TYPE ST_EL3174 :
STRUCT
	Ch1_Error						AT %I*	:BOOL;
	Ch1_Value						AT %I*	:INT;
	Ch2_Error						AT %I*	:BOOL;
	Ch2_Value						AT %I*	:INT;
	Ch3_Error						AT %I*	:BOOL;
	Ch3_Value						AT %I*	:INT;
	Ch4_Error						AT %I*	:BOOL;
	Ch4_Value						AT %I*	:INT;
	State							AT %I*	:UINT;
END_STRUCT
END_TYPE

(* stored: Version 1.1.0.1
   DUT ST_EL3174: Id {723921e4-7ffc-481a-b9b1-e4ad0e9bef43} *)
